{attribute 'linkalways'} 
{attribute 'no_explicit_call' := 'This FB is a CLASS and must be accessed using methods or properties'}
{attribute 'enable_dynamic_creation'}
FUNCTION_BLOCK _LWORD EXTENDS NumericDatatypeBase
VAR
	localData : LWORD;
	activeData : REFERENCE TO LWORD REF= localData;
END_VAR

PROPERTY PUBLIC Address : PVOID
GET
Address := ADR(activeData);
END_GET
END_PROPERTY

METHOD PUBLIC ClearReference
VAR_INPUT
END_VAR
activeData REF= localData;
END_METHOD

METHOD PUBLIC Clone : I_Datatype
VAR
    pClone : POINTER TO _LWORD;
END_VAR
pClone := __NEW(_LWORD(InitialValue := Value));
Clone := pClone^;
END_METHOD

METHOD FB_init : BOOL
VAR_INPUT
	bInitRetains : BOOL; // if TRUE, the retain variables are initialized (warm start / cold start)
	bInCopyCode : BOOL;  // if TRUE, the instance afterwards gets moved WORDo the copy code (online change)
	InitialValue : LWORD;
END_VAR
localData := InitialValue;
END_METHOD

PROPERTY PUBLIC IsFloat : BOOL
GET
IsFloat := FALSE;
END_GET
END_PROPERTY

PROPERTY PUBLIC IsSigned : BOOL
GET
IsSigned := FALSE;
END_GET
END_PROPERTY

METHOD PUBLIC MakeReferenceTo
VAR_INPUT
	ReferenceTarget : REFERENCE TO LWORD;
END_VAR
activeData REF= ReferenceTarget;
END_METHOD

PROPERTY PUBLIC MaxValue : LWORD
GET
MaxValue :=  DatatypeLimits.LWORD_MAX_VALUE;
END_GET
END_PROPERTY

PROPERTY PUBLIC MinValue : LWORD
GET
MinValue := DatatypeLimits.LWORD_MIN_VALUE;
END_GET
END_PROPERTY

METHOD PROTECTED SerializeMaxValue
VAR_INPUT
	Serializer : I_Serializer;
END_VAR
Serializer.AddLword(MaxValue);
END_METHOD

METHOD PROTECTED SerializeMinValue
VAR_INPUT
	Serializer : I_Serializer;
END_VAR
Serializer.AddLword(MinValue);
END_METHOD

METHOD PUBLIC SerializeWith
VAR_INPUT
	Serializer : I_Serializer;
END_VAR
Serializer.AddLword(activeData);
END_METHOD

PROPERTY PUBLIC Size : UDINT
GET
Size := SIZEOF(activeData);
END_GET
END_PROPERTY

METHOD TryDeserializeFrom : BOOL
VAR_INPUT
	Deserializer : I_Deserializer;
	Feedback : I_DeserializerFeedback;
END_VAR
TryDeserializeFrom := Deserializer.TryGetLword(activeData, Feedback);
END_METHOD

METHOD TryMakeReferenceTo : BOOL
VAR_INPUT
	Target : I_Datatype;
END_VAR
VAR
	pTargetData : POINTER TO LWORD;
END_VAR
IF NOT (Target.TypeName = TypeName) THEN
	RETURN;
END_IF

pTargetData := Target.Address;
activeData REF= pTargetData^;
TryMakeReferenceTo := TRUE;
END_METHOD

PROPERTY PUBLIC TypeName : T_MAXSTRING
GET
TypeName := 'LWORD';
END_GET
END_PROPERTY

PROPERTY PUBLIC Value : LWORD
GET
Value := activeData;
END_GET
SET
activeData := Value;
END_SET
END_PROPERTY

END_FUNCTION_BLOCK

(* stored: Version 1.1.0.1, ProductVersion 3.1.4024.12
   POU _LWORD: Id {8aa807cc-58e7-42e6-81e2-6f7e262e8e87}, SpecialFunc None
   Folder Constructor: Id {bb9048a1-4ca3-4a2a-a1d5-cc50ce1772c9}
   Folder Protected: Id {f1603e14-88cb-47b5-b1d5-d1ffa355ca65}
   Property Address: Id {2960a413-15e0-408d-a873-320c8f0fe776}
   Get Get: Id {b8dc27f4-aee3-4eb5-949b-e33a98e8e6e7}
   Method ClearReference: Id {dea7ec8d-dab6-44b6-8789-197451d155a0}
   Method Clone: Id {730f6db4-fbd9-4e90-bdf1-f5d6561cc330}
   Method FB_init: Id {a270308c-63ec-4673-aed9-0c6784024c60}
   Property IsFloat: Id {c4a5c415-df95-47a8-a17a-19081297da32}
   Get Get: Id {78019c08-39c3-4536-87a5-ff1e4d856e56}
   Property IsSigned: Id {85a09bc4-42f1-420e-b5cf-91530c0ebed3}
   Get Get: Id {5686ea2b-be50-4931-9f5c-684e9a221f50}
   Method MakeReferenceTo: Id {f83c2c3d-3f74-48df-be72-ce7884810d0c}
   Property MaxValue: Id {ac5b9b20-8781-41b1-9177-8209227cd2c6}
   Get Get: Id {f1b01f99-af17-4a5b-9506-72d796f946c7}
   Property MinValue: Id {641464d8-bb11-4295-9515-8d96b54006a0}
   Get Get: Id {16ad6c46-eeea-413f-b3ef-6c418e4c1516}
   Method SerializeMaxValue: Id {0421eeeb-1678-45e0-90ae-51e0befa3f0e}
   Method SerializeMinValue: Id {7b3d5558-fc8f-4c1c-97c2-3bccd5c30e05}
   Method SerializeWith: Id {48efaed3-0ea4-4fc5-aba2-10f2f4dedabd}
   Property Size: Id {4b982674-2542-438a-b89e-454927abf449}
   Get Get: Id {d91ad614-220b-47bc-857d-1dfd7c5fe492}
   Method TryDeserializeFrom: Id {1fd0da2f-b65f-40bf-8bdb-6943cca3bbcc}
   Method TryMakeReferenceTo: Id {208dd36b-7539-469a-970d-54718253abfc}
   Property TypeName: Id {a3d93220-67e9-467e-8df8-99efb6aa296a}
   Get Get: Id {baf864d7-1f4b-4027-b196-0f8789947509}
   Property Value: Id {177b8ca6-5e7b-4bc9-89ab-f56395a81e9e}
   Get Get: Id {01e69469-b4d6-4465-9236-4483f5d443e4}
   Set Set: Id {9ceae39a-8436-414d-955b-b354c82babb0} *)
